// SIMATIC S7-200 project (STEP 7-Micro/WIN), CPU 216 REL 01.02

SYMBOL_TABLE SYM1
Always_On        SM0.0    // This bit is always on.
First_Scan_On    SM0.1    // This bit is on for the first scan cycle only.
Pot0_Value       SMB28    // Stores value entered by analog adjustment 0. Updated once per cycle in STOP/RUN
Pot1_Value       SMB29    // Stores value entered by analog adjustment 1. Updated once per cycle in STOP/RUN
Run_Compare      M0.0     // Memory bit must be set to compare the average value to upper and lower limits.
END_SYMBOL_TABLE

ORGANIZATION_BLOCK OB_1:OB1
TITLE=
// ***PROGRAM DESCRIPTION***
// At program startup, initialization is performed during the first scan cycle. The preset time of the fine-tuning mode timer is set to 200ms, while the scan cycle counter is initialized to 0, the working area lower limit memory to 32,000, and the working area upper limit memory to 0, ensuring the correctness of subsequent operations.
// When the user enables fine-tuning mode, a subroutine is called. The value of analog potentiometer 0 is scaled and offset by 200ms, then stored as the preset time for the fine-tuning mode timer. Subsequently, each time the fine-tuning mode timer expires, the subroutine updates the preset time based on the latest value of analog potentiometer 0. Meanwhile, the cycle counter increments and is displayed via the output, allowing the user to monitor the fan's operating status and achieve precise time control.
// If the user enables stable mode, the system samples the value of analog potentiometer 1 100 times through a subroutine, accumulating the results in the accumulator. When the scan cycle counter reaches 100, the subroutine calculates the average value, adjusts it based on the working area lower limit memory and working area upper limit memory, and stores the result in the filtered value memory. This value is then used as the preset time for the stable mode timer. After the timer expires, the cycle counter increments and is displayed via the output, ensuring stable fan runtime and avoiding frequent changes due to potentiometer jitter.
// When the user enables direct load mode and fine-tuning mode is not enabled, the system enters direct load mode. The value of analog potentiometer 0 is directly loaded into the preset time of the direct load mode timer. After timeout, the cycle counter increments and is displayed via the output, allowing real-time adjustment of the fan runtime. However, this value may vary with scan cycles and be less stable.
// 
// 
BEGIN
Network 1 //  First Scan Cycle Initialization
//  Load special memory bit SM0.1 to process this network in the
//  first scan cycle only.
//  Move the constant 0 as an input double word into accumulator AC0
//  to clear the accumulator (set its value to 0).
//  Move the constant 0 as an input double word into accumulator AC2
//  to clear the accumulator (set its value to 0).
//  Move the constant 0 as an input double word into accumulator AC3
//  to clear the accumulator (set its value to 0).
//  Store 20 in variable memory word VW0 to be used as the Preset Time
//  (PT) of timer T33. Timer T33 has a resolution of 10 ms, that is,
//  each count of the current value of timer T33 is a multiple of
//  10 ms. A Preset Time of 20 in this case provides the 200-ms offset
//  needed for option 1.
//  Move the constant 0 as an input word into variable memory word
//  VW10 to set the scan counter for option 2 to 0.
//  Move the constant 32000 as an input word into variable memory word
//  VW14 to reset the lower limit of the workspace.
//  Move the constant 0 as an input word into variable memory word
//  VW16 to reset the upper limit of the workspace.
// 
LD     First_Scan_On:SM0.1   // Load S0.1.
MOVD   +0, AC0               // Clear accumulator AC0.
MOVD   +0, AC2               // Clear accumulator AC2.
MOVD   +0, AC3               // Clear accumulator AC3.
MOVW   +20, VW0              // Store value to be used
// with timer T33.
MOVW   +0, VW10              // Set the scan counter to 0.
MOVW   +32000, VW14          // Reset lower limit
// workspace.
MOVW   +0, VW16              // Reset upper limit
// workspace.
Network 2 //  Option 1
//  The value from an analog potentiometer can vary a few counts each
//  scan cycle. The following logic is used to capture the scaled
//  value from POT0 once per timer cycle, to provide a stable Preset
//  Time for a timer.
// 
//  Load input I0.0 to enable timer T33 and call subroutine SBR1.
//  (This action enables option 1.)
//  Enable timer T33, loading the value in variable memory word VW0
//  from analog adjustment 0 (SMB28, or POT0) as the Preset Time.
//  Call SBR1 to scale and offset the value of analog adjustment 0.
// 
LD     I0.0                  // Load input I0.0.
TON    T33, VW0              // Enable timer T33, with PT
// from VW0.
CALL   SBR_1:SBR1            // Call SBR1.
Network 3 //  Option 1 Continued
//  Load timer T33.
//  If T33 is on (that is, when the current value of the timer = the
//  Preset Time), then increment the value of accumulator AC2 by 1
//  to count the timer cycles.
//  Move (copy) the least significant byte of accumulator AC2 into
//  output byte QB0 to display the number of timer cycles.
//  Reset timer T33.
// 
LD     T33                   // Load timer T33.
INCW   AC2                   // Increment the value of
// accumulator AC2 by 1.
MOVB   AC2, QB0              // Display the current value
// at the output.
R      T33, 1                // Reset timer T33.
Network 4 //  Option 2
//  The value from analog potentiometer POT1 is filtered to provide
//  a constant value for the Preset Time of a timer.
// 
//  Load input I0.1 to call subroutine SBR2 and enable timer T34.
//  (This action enables option 2.)
//  Call subroutine SBR2 to filter the value of analog adjustment 1.
//  Enable timer T34, loading the Preset Time from analog
//  adjustment 1 (SMB29, or POT1)
// 
LD     I0.1                  // Load input I0.1.
CALL   SBR_2:SBR2            // Call SBR2.
TON    T34, VW18             // Enable timer T34, with PT
// from VW18.
Network 5 //  Option 2 Continued
//  Load timer T34.
//  If T34 is on (that is, when the current value of the timer = the
//  Preset Time), then increment the value in variable memory word
//  VW20 by 1 to count the timer cycles.
//  Move (copy) the least significant byte of variable memory word
//  VW20 into output byte QB1 to display the number of timer cycles.
//  Reset timer T34.
// 
LD     T34                   // Load timer T34.
INCW   VW20                  // Increment the value in VW20
// by 1.
MOVB   VB21, QB1             // Display the current value of
// VW20 at the output.
R      T34, 1                // Reset timer T34.
Network 6 //  Option 3
//  The value of POT0 is copied directly to the Preset Time of a timer.
// 
//  Load input I0.2
//  If input I0.2 is on
//  and input I0.0 is not on (this combination enables option 3):
//  move the constant 0 as an input word into accumulator AC1 to
//  clear the accumulator (set its value to 0),
//  move the value in special memory byte SMB28 (analog adjustment 0,
//  or POT0) into accumulator AC1,
//  and enable timer T35, loading the Preset Time from accumulator AC1
//  (that is, the value of analog adjustment 0, or POT0).
// 
LD     I0.2                  // Load input I0.2 as a
// Normally Open contact.
AN     I0.0                  // Handle input I0.0 as a
// Normally Closed contact.
MOVW   +0, AC1               // Clear accumulator AC1.
MOVB   Pot0_Value:SMB28, AC1 // Load analog adjustment 0
// into accumulator AC1.
TON    T35, AC1              // Enable timer T35, with PT
// from AC1.
Network 7 //  Option 3 Continued
//  Load timer T35.
//  If T35 is on (that is, when the current value of the timer = the
//  Preset Time), then increment the value in accumulator AC2 by 1
//  to count the timer cycles.
//  Move (copy) the least significant byte of accumulator AC2 into
//  output byte QB0 to display the number of timer cycles.
//  Reset timer T35.
// 
LD     T35                   // Load timer T35.
INCW   AC2                   // Increment the value in AC2
// by 1.
MOVB   AC2, QB0              // Display the current value
// of AC2 at the output.
R      T35, 1                // Reset timer T35.
Network 8 //  Main Program End
//  End the main program.
//  MEND					// End the main program.
// 
END_ORGANIZATION_BLOCK

SUBROUTINE_BLOCK SBR_1:SBR1
TITLE=
// ***SUBROUTINES***
// 
// 
BEGIN
Network 2 //  Perform the Calculation for Option 1
//  Scale the value of analog adjustment 0 (POT0) and add to an offset
//  which is returned to the main program in VW0.
// 
//  Load timer T33 to check for changes to the analog adjustment 0
//  (POT0) each timer cycle.
//  If T33 is on (that is, when the current value of the timer = the
//  Preset Time):
//  move the constant 0 as an input word into accumulator AC1 to
//  clear the accumulator (set its value to 0),
//  move the value in special memory byte SMB28 (analog adjustment 0,
//  or POT0) into accumulator AC1,
//  move the constant 2 as an input word into variable memory word 60
//  (for compatibility with the ladder logic editor),
//  divide the value of analog adjustment 0 by 2 (to scale the
//  potentiometer input range, which is normally from 0 to 255, by
//  one half: that is, to achieve a scaled range of 0 to 127) and put
//  the result in accumulator AC1,
//  add the constant 20 (for the 200-ms offset) to the value in
//  accumulator AC1 and put the result in accumulator AC1 (this will
//  become the new Preset Time for timer T33),
//  and move the value in accumulator AC1 to variable memory word VW0
//  so that the value can be read by means of a programming device.
// 
LD     T33                   // Load timer T33.
MOVW   +0, AC1               // Clear accumulator AC1.
MOVB   Pot0_Value:SMB28, AC1 // Load analog adjustment 0
// into accumulator AC1.
MOVW   +2, VW60              // Store 2 in VW60.
DIV    VW60, AC1             // Divide the value in AC1 by 2.
+I     +20, AC1              // Add an offset of 200 ms.
MOVW   AC1, VW0              // Move (copy) the value of
// accumulator AC1 to variable
// memory word VW0.
Network 3 //  End of Subroutine SBR1
//  End SBR1. This instruction returns control to the instruction
//  that follows the CALL instruction for SBR1.
//  RET					// End SBR1.
// 
END_SUBROUTINE_BLOCK

SUBROUTINE_BLOCK SBR_2:SBR2
TITLE=
BEGIN
Network 2 //  Count Scan Cycles and Total the Analog Values
//  Sample the value of analog adjustment 1 (POT1) for 100 scan
//  cycles, then get the average value.
// 
//  Load special memory bit SM0.0 to process this network every scan
//  cycle.
//  Increment the value in variable memory word VW10 by 1 to count
//  the scan cycles.
//  Move the value in special memory byte SMB29 (analog adjustment 1,
//  or POT1) into accumulator AC0.
//  Add the value in accumulator AC0 to the value in accumulator AC3
//  (add to the previous total of values from analog adjustment 1).
// 
LD     Always_On:SM0.0       // Load SM0.0.
INCW   VW10                  // Increment the value in VW10
// by 1.
MOVB   Pot1_Value:SMB29, AC0 // Load analog adjustment 1 into
// accumulator AC0.
+I     AC0, AC3              // Add the value in AC0 to the
// value in AC3.
Network 3 //  Calculate Average Analog Value
//  If the value in variable memory word VW10 is equal to 100 (after
//  100 scan cycles):
//  move the constant 100 into variable memory word VW50 (for
//  compatibility with the ladder logic editor),
//  divide the value in accumulator AC3 by 100 (to average the
//  total value),
//  move the value in accumulator AC3 into variable memory word VW12
//  (to save the average value),
//  move the constant 0 into variable memory word VW10 (to reset the
//  scan counter),
//  move the constant 0 as in input double word into accumulator AC3
//  (to reset the work memory for the total of values from SMB29),
//  and turn on memory bit M0.0.
// 
LDW=   VW10, +100            // Compare the value in VW10
// to 100.
MOVW   +100, VW50            // Move 100 into VW50.
DIV    VW50, AC3             // Divide the value in AC3 by 100.
MOVW   AC3, VW12             // Store the result in VW12.
MOVW   +0, VW10              // Move 0 into VW10.
MOVD   +0, AC3               // Move 0 as an input double word
// into AC3.
=      Run_Compare:M0.0      // Turn on M0.0.
Network 4 //  Compare Average Value to Upper and Lower Limits
//  If memory bit M0.0 is on:
//  and the value in variable memory word VW12 (average value of
//  analog adjustment 1) is less than or equal to the value in
//  variable memory word VW14 (lower limit),
//  or the value in variable memory word VW12 (average value of
//  analog adjustment 1) is greater than or equal to the value in
//  variable memory word VW16 (upper limit),
//  fill the memory area starting at VW14 with the word input pattern
//  of VW12 for three words (VW14, VW16, VW18),
//  subtract the constant 3 from the value in variable memory word
//  VW14 and put the result in variable memory word VW14,
//  then add the constant 3 to the value in variable memory word
//  VW16 and put the result in variable memory word VW16.
// 
LD     Run_Compare:M0.0      // Load M0.0.
LDW<=  VW12, VW14            // Compare the value in VW12 to
// the value in VW14 for <=.
OW>=   VW12, VW16            // Compare the value in VW12 to
// the value in VW16 for >=.
ALD                          // Combine the values in the
// first and second levels of
// the stack using a logical And
// operation. Load the result to
// the top of the stack.
FILL   VW12, VW14, 3         // Start at VW14 and fill the
// area with the word input
// pattern of VW12 for three
// words.
-I     +3, VW14              // Subtract 3 from the value
// in VW14.
+I     +3, VW16              // Add 3 to the value in VW16.
Network 5 //  End Subroutine SBR2
//  End SBR2. This instruction returns control to the instruction
//  that follows the CALL instruction for SBR2. This action returns
//  the filtered potentiometer value in variable memory word VW18.
//  RET					// End SBR2.
// 
END_SUBROUTINE_BLOCK
